{attribute addProperty BoxType "EL1258-0000-0017"}
{attribute addProperty Id "StatusAT %I*Status_8577222D3241InputsAT %I*Inputs_8B7B380032433Input_event_timeAT %I*ARRAY[0 ..9] OF UDINT320400"}
{attribute addProperty CRC "3439144347"}
{attribute addProperty SizeInBites "384"}
{attribute addProperty SizeInBytes "48"}
TYPE MTI_Inputs_10x_Channel_7752F308 :
STRUCT
	{attribute addProperty Name "Status"}
	Status AT %I* : Status_8577222D;
	{attribute addProperty Name "Inputs"}
	Inputs AT %I* : Inputs_8B7B3800;
	{attribute addProperty Name "Input_event_time"}
	Input_event_time AT %I* : ARRAY[0 ..9] OF UDINT;
END_STRUCT
END_TYPE

(* stored: Version 1.2.0.0, ProductVersion 3.1.4024.9
   DUT MTI_Inputs_10x_Channel_7752F308: Id {a5c538ca-52c7-46d6-ba5d-4bb67083649f} *)
